# B&R Automation Studio project Vrtalka
Automation Studio 4.2.10.53 SP

## Configuration HW_config

### Task classes (Cpu.sw)
```
Cyclic#4 (cycle 100000 us, tolerance 100000 us):
  Vrtalka <- Vrtalka.prg
VcDataObjects: Vrtalk <- HMI.VrtalkaHMI.dob
```

### Hardware
```
4PPC70_101G_20B : 4PPC70.101G-20B v1.4.0.0
  Connector IF2:
    ActivateDevice = 1
    HostName = arsim
    Vnc1
    VncKeyMappingFile1 = VC\PS2-Keyboard1.dis
    VncMaxConnections1 = 2
    VncRefreshRate1 = 100
    VncTitle1 = HMIvrt
  ConfigurationID = Vrtalka_HW_config
  Simulation = 1
  Connections = 5
  TimerDeviceType = SWIOTIMER
  Cyclic1Duration = 10000
  Cyclic1Tolerance = 10000
  Cyclic2Duration = 20000
  Cyclic2Tolerance = 20000
  Cyclic3Duration = 50000
  Cyclic3Tolerance = 50000
  Cyclic4Duration = 100000
  Cyclic4Tolerance = 100000
  Cyclic5Duration = 200000
  Cyclic5Tolerance = 200000
  Cyclic6Duration = 500000
  Cyclic6Tolerance = 500000
  Cyclic7Duration = 1000000
  Cyclic7Tolerance = 1000000
  Cyclic8Duration = 10000
  Cyclic8Tolerance = 30000000
  VcObjectName = Vrtalk
  KeyMappingFile = VC\4PPC70_101G_20B.dis
```

## Configuration SimConf

CPU 4PPC70.101G-20B, AutomationRuntime D4.26, Build 4.1.2, Vc V4.26.5

### Task classes (Cpu.sw)
```
Cyclic#4:
  programHMI <- HMI.programHMI.prg [disabled]
Cyclic#7:
  Vrtalka <- Vrtalka.prg [disabled]
VcDataObjects: Vrtalk <- HMI.VrtalkaHMI.dob
Binaries: vcfile, vcrt, vctcal, vcfntttf, vcctext, arial, vcalarm, vcmgr, vccovl, vccnum, vcpfar00, vcdsint, vcpdvnc, vccslider, vcshared, vcpdsw, seguisb, vccbtn, Vrtalk03, vccstr, vcgclass, vcdsloc, arialbd, vcnet, TCData, segoeuib, segoeui, vccbmp, vcbclass, vccline, solid4n6, Vrtalk02, Vrtalk01, vccshape, User, ashwd, arconfig, sysconf, Role, asfw, iomap, Vrtal103, Vrtal102, vcpkat
Libraries: fileio, asieccon, dataobj, vcresman, astime, runtime
```

## Configuration SimulationConfig

CPU 4PPC70.101G-20B, AutomationRuntime D4.26, Build 4.1.2, Vc V4.26.5

### Task classes (Cpu.sw)
```
Cyclic#4 (cycle 100000 us, tolerance 100000 us):
  Program <- Program.prg
VcDataObjects: Vrtalk <- VrtalkaHMI.dob
Binaries: vcmgr, vcpfar00, arialbd, vcpdsw, vcalarm, vcshared, vcnet, vcgclass, vctcal, Vrtalk01, TCData, vcpdvnc, vccnum, Vrtalk02, vcfntttf, vcctext, Vrtalk03, vcdsint, vcfile, vcpkat, vcrt, vcbclass, vcdsloc, vccovl, arial, vccslider, vccbtn, reemkz6g, vccbmp, vccline, ashwd, User, sysconf, asfw, arconfig, iomap, Role, vccbar
Libraries: MTBasics, brsystem, MTTypes, sys_lib, runtime, fileio, vcresman, dataobj, asieccon, astime
```

### Hardware
```
4PPC70_101G_20B : 4PPC70.101G-20B v1.4.0.0
  Connector IF2:
    ActivateDevice = 1
    HostName = vrtalkahmi
    Vnc1
    VncVcObjectName1 = Vrtalk
    VncKeyMappingFile1 = VC\PS2-Keyboard.dis
    VncRefreshRate1 = 100
    VncTitle1 = Vrtalka
  ConfigurationID = Vrtalka_Config1
  TimerDeviceType = SWIOTIMER
  Cyclic1Duration = 10000
  Cyclic1Tolerance = 10000
  Cyclic2Duration = 20000
  Cyclic2Tolerance = 20000
  Cyclic3Duration = 50000
  Cyclic3Tolerance = 50000
  Cyclic4Duration = 100000
  Cyclic4Tolerance = 100000
  Cyclic5Duration = 200000
  Cyclic5Tolerance = 200000
  Cyclic6Duration = 500000
  Cyclic6Tolerance = 500000
  Cyclic7Duration = 1000000
  Cyclic7Tolerance = 1000000
  Cyclic8Duration = 10000
  Cyclic8Tolerance = 30000000
  KeyMappingFile = VC\4PPC70_101G_20B.dis
```

## Logical view

Binary libraries used (declarations not repeated): operator, runtime, astime, AsIecCon, MTBasics 2.30.0, brsystem, MTTypes 1.03.4, sys_lib


### Program Logical/Vrtalka (IEC)

#### AGR_Actions.st
```iecst
ACTION SomeTestAction:
	diHMIin2 := TRUE;
END_ACTION

ACTION SetInitialAgrValues:
	// Nastavi sirine agregatov
	agr1.agr_width := 30;
	agr2.agr_width := 30;
	agr3.agr_width := 30;
	agr4.agr_width := 30;
	agr5.agr_width := 30;
	agr6.agr_width := 30;

	// Nastavi minimalne pozicje agregatov
	agr1.poz_agr_min := agr1.agr_width;
	agr2.poz_agr_min := agr1.poz_agr_min + agr2.agr_width;
	agr3.poz_agr_min := agr2.poz_agr_min + agr3.agr_width;
	agr4.poz_agr_min := agr3.poz_agr_min + agr4.agr_width;
	agr5.poz_agr_min := agr4.poz_agr_min + agr5.agr_width;
	agr6.poz_agr_min := agr5.poz_agr_min + agr6.agr_width;

	// Reset nastavljenih pozicj
	agr1.poz_agr_s := 0;
	agr2.poz_agr_s := 0;
	agr3.poz_agr_s := 0;
	agr4.poz_agr_s := 0;
	agr5.poz_agr_s := 0;
	agr6.poz_agr_s := 0;

	// Reset trenutnih pozicij
	agr1.poz_agr_a := 0;
	agr2.poz_agr_a := 0;
	agr3.poz_agr_a := 0;
	agr4.poz_agr_a := 0;
	agr5.poz_agr_a := 0;
	agr6.poz_agr_a := 0;

	// Reset okej boolov
	agr1.agr_pos_ok := FALSE;
	agr2.agr_pos_ok := FALSE;
	agr3.agr_pos_ok := FALSE;
	agr4.agr_pos_ok := FALSE;
	agr5.agr_pos_ok := FALSE;
	agr6.agr_pos_ok := FALSE;

	// Reset ali je agr aktiven
	agr1.agr_active := FALSE;
	agr2.agr_active := FALSE;
	agr3.agr_active := FALSE;
	agr4.agr_active := FALSE;
	agr5.agr_active := FALSE;
	agr6.agr_active := FALSE;

	// Nastavi status agregata
	agr1.ag_status := 0;
	agr2.ag_status := 0;
	agr3.ag_status := 0;
	agr4.ag_status := 0;
	agr5.ag_status := 0;
	agr6.ag_status := 0;

END_ACTION

ACTION SetMaxAgrValues:  (* Izracun trenutnih maksimalnih pozicij *)

END_ACTION

// Sprosti zavore na agregatih
ACTION ReleaseAgrBrakes:
	ZavoraAgregata(agr1, FALSE);
	ZavoraAgregata(agr2, FALSE);
	ZavoraAgregata(agr3, FALSE);
	ZavoraAgregata(agr4, FALSE);
	ZavoraAgregata(agr5, FALSE);
	ZavoraAgregata(agr6, FALSE);

END_ACTION

ACTION LockAgrBrakes:
	ZavoraAgregata(agr1, TRUE);
	ZavoraAgregata(agr2, TRUE);
	ZavoraAgregata(agr3, TRUE);
	ZavoraAgregata(agr4, TRUE);
	ZavoraAgregata(agr5, TRUE);
	ZavoraAgregata(agr6, TRUE);

END_ACTION

ACTION SetHomePosAgr: (* Vse agregate peljemo na minimalne pozicije *)
	(*
	Nastaviti se morajo naslednje spremenljivke
	agr<#>.poz_agr_s - vozicke prepeljemo v minimalne lege dolocene v spremenljivki agr<#>.poz_agr_min
	agr<#>.poz_agr_a - dejanske pozicije agregatov (agregati so skupaj in naslonjeni, izracuna se iz sirine agregatov)
	agr<#>.poz_agr_i - izhodiscna pozicija agregata, ce zelimo kasneje popraviti lego, peljemo v HOME in nazaj razporedimo
	*)
	// Pomaknemo vozicek v max ce se ni
	PomikVozicka(1000, vozicek);
	// Iztegnemo zaklep na vozicku
	ZaklepAgregata(vozicek, TRUE);
	// Pomaknemo vozicek iz maksimuma v minimalno lego agregata 6 - agregati se med seboj dotikajo)
	PomikVozicka(agr6.poz_agr_min, vozicek);

	// Nastavimo status vozicka
	agr1.ag_status := 3;
	agr2.ag_status := 3;
	agr3.ag_status := 3;
	agr4.ag_status := 3;
	agr5.ag_status := 3;
	agr6.ag_status := 3;

	// Pozicije agregatov so sedaj znane
	// Agr1
	agr1.ag_status := 2;
	agr1.poz_agr_s := agr1.poz_agr_min;
	agr1.poz_agr_a := agr1.poz_agr_s;
	agr1.poz_agr_i := agr1.poz_agr_a;
	agr1.agr_pos_ok := TRUE;
	// Agr 2
	agr2.ag_status := 2;
	agr2.poz_agr_s := agr2.poz_agr_min;
	agr2.poz_agr_a := agr2.poz_agr_s;
	agr2.poz_agr_i := agr2.poz_agr_a;
	agr2.agr_pos_ok := TRUE;
	// Agr 3
	agr3.ag_status := 2;
	agr3.poz_agr_s := agr3.poz_agr_min;
	agr3.poz_agr_a := agr3.poz_agr_s;
	agr3.poz_agr_i := agr3.poz_agr_a;
	agr3.agr_pos_ok := TRUE;
	// Agr 4
	agr4.ag_status := 2;
	agr4.poz_agr_s := agr4.poz_agr_min;
	agr4.poz_agr_a := agr4.poz_agr_s;
	agr4.poz_agr_i := agr4.poz_agr_a;
	agr4.agr_pos_ok := TRUE;
	// Agr 5
	agr5.ag_status := 2;
	agr5.poz_agr_s := agr5.poz_agr_min;
	agr5.poz_agr_a := agr5.poz_agr_s;
	agr5.poz_agr_i := agr5.poz_agr_a;
	agr5.agr_pos_ok := TRUE;
	// Agr 6
	agr6.ag_status := 2;
	agr6.poz_agr_s := agr6.poz_agr_min;
	agr6.poz_agr_a := agr6.poz_agr_s;
	agr6.poz_agr_i := agr6.poz_agr_a;
	agr6.agr_pos_ok := TRUE;

END_ACTION

ACTION SetIzbraniAgrVal: (* Nastavljanje spremenljivke izbrani_agr iz boolov aktivnih agr *)

	// Za vsak agregat se preveri ce je aktiviran in ce je ustrezen bit v spremenljivki izbrani_agr postavljen na 1
	IF (agr1.agr_active = TRUE) AND (izbrani_agr.0 = 0) THEN
		izbrani_agr.0 := 1;
	ELSIF (agr1.agr_active = FALSE) AND (izbrani_agr.0 = 1) THEN
		izbrani_agr.0 := 0;
	END_IF;

	IF (agr2.agr_active = TRUE) AND (izbrani_agr.1 = 0) THEN
		izbrani_agr.1 := 1;
	ELSIF (agr2.agr_active = FALSE) AND (izbrani_agr.1 = 1) THEN
		izbrani_agr.1 := 0;
	END_IF;

	IF (agr3.agr_active = TRUE) AND (izbrani_agr.2 = 0) THEN
		izbrani_agr.2 := 1;
	ELSIF (agr3.agr_active = FALSE) AND (izbrani_agr.2 = 1) THEN
		izbrani_agr.2 := 0;
	END_IF;

	IF (agr4.agr_active = TRUE) AND (izbrani_agr.3 = 0) THEN
		izbrani_agr.3 := 1;
	ELSIF (agr4.agr_active = FALSE) AND (izbrani_agr.3 = 1) THEN
		izbrani_agr.3 := 0;
	END_IF;

	IF (agr5.agr_active = TRUE) AND (izbrani_agr.4 = 0) THEN
		izbrani_agr.4 := 1;
	ELSIF (agr5.agr_active = FALSE) AND (izbrani_agr.4 = 1) THEN
		izbrani_agr.4 := 0;
	END_IF;

	IF (agr6.agr_active = TRUE) AND (izbrani_agr.5 = 0) THEN
		izbrani_agr.5 := 1;
	ELSIF (agr6.agr_active = FALSE) AND (izbrani_agr.5 = 1) THEN
		izbrani_agr.5 := 0;
	END_IF;

END_ACTION
```

#### SRV_Actions.st
```iecst
ACTION SetInitialSrvValues:
	// Relevatne vrednosti pozicij
	vozicek.poz_srv_max := 1000;
	vozicek.poz_srv_min := agr1.poz_agr_min;

	// Reset ostalih spremenljivk

	// Zaklep agregata noter (Varnost)
	ZaklepAgregata(vozicek, FALSE);
	TestZaklepaAgr(vozicek);

	vozicek.servo_act := 0;
	vozicek.servo_set := 0;

	vozicek.servo_in_pos := FALSE;
	vozicek.servo_moving := FALSE;

	// Zaklep agregata noter ter pomik v skrajno lego
	PomikVozicka(n_pos := vozicek.poz_srv_max, vozicek := vozicek);
END_ACTION
```

#### General_actions.st
```iecst
ACTION ReadVarsFromHMI: (* Preberi vse spremenljivke iz HMI ekrana *)
	// Dummy
	diHMIin1 := diHMIin1;

	// Agregat
	agr1.agr_active := agr1.agr_active;
	agr2.agr_active := agr2.agr_active;
	agr3.agr_active := agr3.agr_active;
	agr4.agr_active := agr4.agr_active;
	agr5.agr_active := agr5.agr_active;
	agr6.agr_active := agr6.agr_active;

	SetIzbraniAgrVal;

	agr1.poz_agr_s := agr1.poz_agr_s;
	agr2.poz_agr_s := agr2.poz_agr_s;
	agr3.poz_agr_s := agr3.poz_agr_s;
	agr4.poz_agr_s := agr4.poz_agr_s;
	agr5.poz_agr_s := agr5.poz_agr_s;
	agr6.poz_agr_s := agr6.poz_agr_s;

END_ACTION
```

#### PROC_actions.st
```iecst
ACTION makeStep:
	WHILE diSTEP = FALSE DO
	END_WHILE;
	diSTEP := FALSE;
END_ACTION

ACTION nastavljanjeAgregatov:

	// Preveri ce so vse pozicije agregatov znane
	diPozAgrOK := agr1.agr_pos_ok AND agr2.agr_pos_ok AND agr3.agr_pos_ok AND agr4.agr_pos_ok AND agr5.agr_pos_ok AND agr6.agr_pos_ok;
	SetIzbraniAgrVal;
	makeStep;
	IF diPozAgrOK = FALSE THEN
		SetHomePosAgr;
	END_IF;
	makeStep;
	IF currentPage <> 20 THEN
		changePage := 20;
	END_IF;

	makeStep;

	// Pocakaj za vsak slucaj da se odpre nastavitven ekran
	WHILE currentPage <> 20 DO
	END_WHILE;
	sistemskoObvestilo := 'Stroj v nastavljanju';

	WHILE diShraniPozicije = FALSE DO
	END_WHILE;
	ReadVarsFromHMI;
	popupConfirm := 0;

	WHILE diPotrdiPozicije = FALSE DO
	END_WHILE;

	diShraniPozicije := FALSE;
	diPotrdiPozicije := FALSE;
	popupConfirm := 1;

	// Stroj je pripravljen na delo, nastavitve agregatov so potrjene
	// Stroj je priprvljen na uporabo
	doStrojPripravljen := TRUE;

	WHILE diStartStroja = FALSE DO
	END_WHILE;

	//popupWarning := 1;
	changePage := 10;

END_ACTION

ACTION OperacijaVrtanja: (* mock operacija za vrtanje *)
	// Tukaj bi prisla koda za dejansko vrtanje vrtalke
END_ACTION
```

#### Cyclic.st - Cyclic code
```iecst
PROGRAM _CYCLIC
	// Preveri ali je stroj pripravljen na delovanje
	IF doStrojPripravljen = FALSE THEN
		nastavljanjeAgregatov;
	ELSIF (diStartStroja = TRUE OR doDelovanje = TRUE) AND doStrojPripravljen = TRUE THEN
		sistemskoObvestilo := 'Stroj v delovanju';
		doDelovanje := TRUE;
		diStartStroja := FALSE;
		OperacijaVrtanja;
	ELSIF diPrekiniCikel = TRUE AND doDelovanje = TRUE THEN
		sistemskoObvestilo := 'Stroj v zaustavljanju';
		OperacijaVrtanja;
		doDelovanje := FALSE;
		sistemskoObvestilo := 'Stroj zaustavljen';
	END_IF;

END_PROGRAM
```

#### Init.st - Init code
```iecst
PROGRAM _INIT

	//Nastavi trenutno stran na Settings ob zagonu
	changePage := 0;
	sistemskoObvestilo := 'ZAGON STROJA';
	// Resetiraj pozicije in spremenljivke agregatov
	SetInitialAgrValues;
	ReleaseAgrBrakes;
	WHILE diGoHome = FALSE DO
	END_WHILE;

	// Zapri okno
	popupWarning := 1;
	// Resetiraj spremenljivke vozicka in ga zapelji v max lego
	SetInitialSrvValues;
	// Postavi agregate v HOME pozicijo
	SetHomePosAgr;
	diGoHome := FALSE;
END_PROGRAM
```

#### HMIVars.var
```iecst
VAR
	setupScreen : BOOL := FALSE; (*Ali je setup screen aktiven*)
END_VAR
```

### VrtalkaVars.var - Local variables
```iecst
(*Delovne variable*)
VAR
	sistemskoObvestilo : STRING[80] := 'Ni obvestil'; (*spremenljivka za obvestila*)
END_VAR
(*HMI variable*)
VAR
	changePage : UINT := 0; (*spremenljivka za prikaz popupa*)
	popupConfirm : UINT := 0; (*Spremenljivka za pop-up okno ob potrditvi*)
	popupWarning : UINT := 0; (*Spremenljivka za pop-up okno ob zagonu*)
END_VAR
VAR CONSTANT
	settingsPage : UINT := 20; (*Index nastavitvene strani*)
END_VAR
VAR
	currentPage : UINT := 0; (*Spremenljivka ali je setupScreen aktiven*)
END_VAR
(*Agregati*)
VAR
	agr1 : agr_typ := (izbrani_agr_mask:=1); (*agregat 1*)
	agr2 : agr_typ := (izbrani_agr_mask:=2); (*agregat 2*)
	agr3 : agr_typ := (izbrani_agr_mask:=4); (*agregat 3*)
	agr4 : agr_typ := (izbrani_agr_mask:=8); (*agregat 4*)
	agr5 : agr_typ := (izbrani_agr_mask:=16); (*agregat 5*)
	agr6 : agr_typ := (izbrani_agr_mask:=32); (*agregat 6*)
	diPozAgrOK : BOOL; (*ali so pozicije agregatov znane*)
	diHMIin1 : BOOL := FALSE;
	diHMIin2 : BOOL := FALSE;
END_VAR
(*GhostVars [DI/DO]*)
VAR
	diSTEP : BOOL := FALSE; (*Spremenljivka za step-anje*)
	diPrekiniCikel : BOOL := FALSE; (*Prekinitev cikla*)
	diSoftStop : BOOL := FALSE; (*ustavitev delovanja*)
	diStartStroja : BOOL := FALSE; (*digital input za start Stroja*)
	doDelovanje : BOOL := FALSE; (*stroj je v delovanju*)
	diRand : BOOL := FALSE; (*DI random*)
	diSetAgrPoz : BOOL := FALSE; (*DI za pomik agregatov v nastavljene pozicije*)
	diGoHome : BOOL := FALSE; (*DI za homing vozickov -> poz_agr_min*)
	doFunSuccess : BOOL := FALSE; (*Mock HMI prikaz *)
	doHMIout1 : BOOL := FALSE;
	diPotrdiPozicije : BOOL := FALSE; (*shrani in potrdi pozicije*)
	diShraniPozicije : BOOL := FALSE; (*potrdi pozicije agregatov*)
	doStrojPripravljen : BOOL := FALSE; (*stroj je pripravljen za delo*)
	izbrani_agr : UINT := 0; (*int izbranih agregatov*)
END_VAR
(*Nastavljene pozicije agregatov [REAL/D]*)
VAR
	poz_agr_i : REAL := 0.0; (*Skupna sirina agregatov -> izracuna iz st. agregatov in njihove sirine*)
END_VAR
(*Agregati varnostne spemenljivke [REAL]*)
VAR CONSTANT
	raz_agr : REAL := 30; (*Minimalen razmik agregatov, izhaja iz sirine agregatov*)
END_VAR
(*Servo*)
VAR
	vozicek : servo_typ := (0); (*Spremenljivka za servo typ*)
END_VAR
```

### Types.typ
```iecst
TYPE
	agr_typ : 	STRUCT
		poz_agr_s : REAL := 0; (*Nastavljena pozicija agregata*)
		poz_agr_a : REAL := 0; (*Dejanska pozicija agregata*)
		poz_agr_i : REAL; (*Izhodiscna pozicija agregata*)
		poz_agr_min : REAL := 0; (*Minimalna skrajna lega agregata*)
		poz_agr_max : REAL := 0; (*Maksimalna skrajna lega agregata*)
		agr_pos_ok : BOOL := FALSE; (*Agregat v poziciji*)
		o_agr_zav : BOOL := FALSE; (*Zavora agregata*)
		agr_width : REAL := 30; (*Sirina agregata*)
		agr_active : BOOL := FALSE; (*Ali je agregat aktiven*)
		izbrani_agr_mask : UINT; (*Maska za spremenljivko izbrani agregat*)
		ag_status : UINT;
	END_STRUCT;
	servo_typ : 	STRUCT
		servo_set : REAL := 0; (*Nastavljena pozicija servo motorja*)
		servo_act : REAL := 0; (*Trenutna pozicija servo motorja*)
		servo_in_pos : BOOL := FALSE; (*Servo na poziciji*)
		o_agr_zak_z : BOOL := FALSE; (*Razmik agr. -> zaklep ZUNAJ ; OUTPUT*)
		o_agr_zak_o : BOOL := FALSE; (*Razmik agr. -> zaklep NOTER ; OUTPUT*)
		i_agr_zak_z : BOOL := FALSE; (*Razmik agr. -> zaklep ZUNAJ ; INPUT*)
		i_agr_zak_o : BOOL := FALSE; (*Razmik agr. -> zaklep NOTER ; INPUT*)
		poz_srv_max : REAL := 1000; (*Maksimalna pozicija servota*)
		poz_srv_min : REAL := 0; (*Minimalna pozicija servota*)
		servo_moving : BOOL := FALSE; (*DO da se servo premika*)
		agr_zak : BOOL := FALSE; (*ali je agregat zaklnjen (TRUE je, FALSE ni)*)
	END_STRUCT;
END_TYPE
```

- Visualisation Logical/HMI/VrtalkaHMI (not shown)

### Program Logical/HMI/programHMI (IEC)

#### Main.st - Init, cyclic, exit code
```iecst
PROGRAM _INIT
	(* Insert code here *)
	//obvestiloHMI := 'INIT UFNKCIJA';
	popupWarning := 0;
	WHILE diGoHome = FALSE DO
	END_WHILE;
	changePage := 20;
	// Zapri okno
	popupWarning := 1;
END_PROGRAM

PROGRAM _CYCLIC
	(* Insert code here *)
	//obvestiloHMI := 'CIKLIK';
	(* Insert code here *)
	//poz_agr1_a := poz_agr1_a + 5;
	stevec := stevec + 1;
	//changePage := 10;
	ReadVarsFromHMI;

END_PROGRAM

PROGRAM _EXIT
	(* Insert code here *)
	obvestiloHMI := 'ENDER';

END_PROGRAM
```

#### Variables.var - Local variables
```iecst
VAR
	obvestiloHMI : STRING[80] := 'prazno';
	stevec : UINT := 0;
END_VAR
```

#### HMI_actions.st
```iecst
ACTION ReadVarsFromHMI: (* Preberi vse spremenljivke iz HMI ekrana *)
	// Dummy
	diHMIin1 := diHMIin1;

	// Agregat
	agr1 := agr1;
	agr2 := agr2;
	agr3 := agr3;
	agr4 := agr4;
	agr5 := agr5;
	agr6 := agr6;

	diPozAgrOK := diPozAgrOK;

	diSTEP := diSTEP;
	diPrekiniCikel := diPrekiniCikel;
	diSoftStop := diSoftStop;
	diStartStroja := diStartStroja;
	doDelovanje := doDelovanje;
	diRand := diRand;
	diSetAgrPoz := diSetAgrPoz;
	diGoHome := diGoHome;
	doFunSuccess := doFunSuccess;
	doHMIout1 := doHMIout1;
	diPotrdiPozicije := diPotrdiPozicije;
	diShraniPozicije := diShraniPozicije;
	doStrojPripravljen := doStrojPripravljen;
	izbrani_agr := izbrani_agr;

	vozicek := vozicek;

	diHMIin1 := diHMIin1;
	diHMIin2 := diHMIin2;

	(*
	agr1.agr_active := agr1.agr_active;
	agr2.agr_active := agr2.agr_active;
	agr3.agr_active := agr3.agr_active;
	agr4.agr_active := agr4.agr_active;
	agr5.agr_active := agr5.agr_active;
	agr6.agr_active := agr6.agr_active;

	agr1.poz_agr_s := agr1.poz_agr_s;
	agr2.poz_agr_s := agr2.poz_agr_s;
	agr3.poz_agr_s := agr3.poz_agr_s;
	agr4.poz_agr_s := agr4.poz_agr_s;
	agr5.poz_agr_s := agr5.poz_agr_s;
	agr6.poz_agr_s := agr6.poz_agr_s;
	*)
END_ACTION
```

### hmiVariables.var - not listed in the package file held
```iecst
VAR
	hmiPageVar : USINT := 10;
END_VAR
```

### Program Logical/Program (IEC)

#### Variables.var - Local variables
```iecst
(*Delovne variable*)
(*Agregati*)
VAR
	agr1 : agr_typ := (izbrani_agr_mask:=1); (*agregat 1*)
	agr2 : agr_typ := (izbrani_agr_mask:=2); (*agregat 2*)
	agr3 : agr_typ := (izbrani_agr_mask:=4); (*agregat 3*)
	agr4 : agr_typ := (izbrani_agr_mask:=8); (*agregat 4*)
	agr5 : agr_typ := (izbrani_agr_mask:=16); (*agregat 5*)
	agr6 : agr_typ := (izbrani_agr_mask:=32); (*agregat 6*)
	diHMIin1 : BOOL := FALSE;
	diHMIin2 : BOOL := FALSE;
END_VAR
(*GhostVars [DI/DO]*)
VAR
	diPrekiniCikel : BOOL := FALSE; (*Prekinitev cikla*)
	diSoftStop : BOOL := FALSE; (*ustavitev delovanja*)
	diStartStroja : BOOL := FALSE; (*digital input za start Stroja*)
	doDelovanje : BOOL := FALSE; (*stroj je v delovanju*)
	diRand : BOOL := FALSE; (*DI random*)
	diSetAgrPoz : BOOL := FALSE; (*DI za pomik agregatov v nastavljene pozicije*)
	diGoHome : BOOL := FALSE; (*DI za homing vozickov -> poz_agr_min*)
	doFunSuccess : BOOL := FALSE; (*Mock HMI prikaz *)
	doHMIout1 : BOOL := FALSE;
	doStrojPripravljen : BOOL := FALSE; (*stroj je pripravljen za delo*)
	izbrani_agr : UINT := 0; (*int izbranih agregatov*)
END_VAR
(*Nastavljene pozicije agregatov [REAL/D]*)
VAR
	poz_agr_i : REAL := 0.0; (*Skupna sirina agregatov -> izracuna iz st. agregatov in njihove sirine*)
END_VAR
(*Agregati varnostne spemenljivke [REAL]*)
VAR CONSTANT
	raz_agr : REAL := 30; (*Minimalen razmik agregatov, izhaja iz sirine agregatov*)
END_VAR
(*Servo*)
VAR
	vozicek : servo_typ := (0); (*Spremenljivka za servo typ*)
END_VAR
```

#### Types.typ
```iecst
TYPE
	agr_typ : 	STRUCT
		poz_agr_s : REAL := 0; (*Nastavljena pozicija agregata*)
		poz_agr_a : REAL := 0; (*Dejanska pozicija agregata*)
		poz_agr_min : REAL := 0; (*Minimalna skrajna lega agregata*)
		poz_agr_max : REAL := 0; (*Maksimalna skrajna lega agregata*)
		agr_pos_ok : BOOL := FALSE; (*Agregat v poziciji*)
		o_agr_zav : BOOL := FALSE; (*Zavora agregata*)
		agr_width : REAL := 30; (*Sirina agregata*)
		agr_active : BOOL := FALSE; (*Ali je agregat aktiven*)
		izbrani_agr_mask : UINT; (*Maska za spremenljivko izbrani agregat*)
	END_STRUCT;
	servo_typ : 	STRUCT
		servo_set : REAL := 0; (*Nastavljena pozicija servo motorja*)
		servo_act : REAL := 0; (*Trenutna pozicija servo motorja*)
		servo_in_pos : BOOL := FALSE; (*Servo na poziciji*)
		o_agr_zak_z : BOOL := FALSE; (*Razmik agr. -> zaklep ZUNAJ ; OUTPUT*)
		o_agr_zak_o : BOOL := FALSE; (*Razmik agr. -> zaklep NOTER ; OUTPUT*)
		i_agr_zak_z : BOOL := FALSE; (*Razmik agr. -> zaklep ZUNAJ ; INPUT*)
		i_agr_zak_o : BOOL := FALSE; (*Razmik agr. -> zaklep NOTER ; INPUT*)
		poz_srv_max : REAL := 1000; (*Maksimalna pozicija servota*)
		poz_srv_min : REAL := 0; (*Minimalna pozicija servota*)
		servo_moving : BOOL := FALSE; (*DO da se servo premika*)
		agr_zak : BOOL := FALSE; (*ali je agregat zaklnjen (TRUE je, FALSE ni)*)
	END_STRUCT;
END_TYPE
```

#### AGR_Actions.st
```iecst
ACTION SomeTestAction:
	diHMIin2 := TRUE;
END_ACTION

ACTION SetInitialAgrValues:
	// Nastavi sirine agregatov
	agr1.agr_width := 30;
	agr2.agr_width := 30;
	agr3.agr_width := 30;
	agr4.agr_width := 30;
	agr5.agr_width := 30;
	agr6.agr_width := 30;

	// Nastavi minimalne pozicje agregatov
	agr1.poz_agr_min := agr1.agr_width;
	agr2.poz_agr_min := agr1.poz_agr_min + agr2.agr_width;
	agr3.poz_agr_min := agr2.poz_agr_min + agr3.agr_width;
	agr4.poz_agr_min := agr3.poz_agr_min + agr4.agr_width;
	agr5.poz_agr_min := agr4.poz_agr_min + agr5.agr_width;
	agr6.poz_agr_min := agr5.poz_agr_min + agr6.agr_width;

	// Reset nastavljenih pozicj
	agr1.poz_agr_s := 0;
	agr2.poz_agr_s := 0;
	agr3.poz_agr_s := 0;
	agr4.poz_agr_s := 0;
	agr5.poz_agr_s := 0;
	agr6.poz_agr_s := 0;

	// Reset trenutnih pozicij
	agr1.poz_agr_a := 0;
	agr2.poz_agr_a := 0;
	agr3.poz_agr_a := 0;
	agr4.poz_agr_a := 0;
	agr5.poz_agr_a := 0;
	agr6.poz_agr_a := 0;

	// Reset okej boolov
	agr1.agr_pos_ok := FALSE;
	agr2.agr_pos_ok := FALSE;
	agr3.agr_pos_ok := FALSE;
	agr4.agr_pos_ok := FALSE;
	agr5.agr_pos_ok := FALSE;
	agr6.agr_pos_ok := FALSE;

	// Reset ali je agr aktiven
	agr1.agr_active := FALSE;
	agr2.agr_active := FALSE;
	agr3.agr_active := FALSE;
	agr4.agr_active := FALSE;
	agr5.agr_active := FALSE;
	agr6.agr_active := FALSE;

END_ACTION

ACTION SetMaxAgrValues:  (* Izracun trenutnih maksimalnih pozicij *)

END_ACTION

// Sprosti zavore na agregatih
ACTION ReleaseAgrBrakes:
	ZavoraAgregata(agr1, FALSE);
	ZavoraAgregata(agr2, FALSE);
	ZavoraAgregata(agr3, FALSE);
	ZavoraAgregata(agr4, FALSE);
	ZavoraAgregata(agr5, FALSE);
	ZavoraAgregata(agr6, FALSE);

END_ACTION

ACTION SetHomePosAgr: (* Vse agregate peljemo na minimalne pozicije *)
	// Pomaknemo vozicek v max ce se ni
	PomikVozicka(1000, vozicek);
	// Iztegnemo zaklep na vozicku
	ZaklepAgregata(vozicek, TRUE);
	// Pomaknemo vozicek iz maksimuma v minimalno lego agregata 6 - agregati se med seboj dotikajo)
	PomikVozicka(agr6.poz_agr_min, vozicek);

	// Pozicije agregatov so sedaj znane
	// Agr1
	agr1.poz_agr_s := agr1.poz_agr_min;
	agr1.poz_agr_a := agr1.poz_agr_min;
	agr1.agr_pos_ok := TRUE;
	// Agr 2
	agr2.poz_agr_s := agr2.poz_agr_min;
	agr2.poz_agr_a := agr2.poz_agr_min;
	agr2.agr_pos_ok := TRUE;
	// Agr 3
	agr3.poz_agr_s := agr3.poz_agr_min;
	agr3.poz_agr_a := agr3.poz_agr_min;
	agr3.agr_pos_ok := TRUE;
	// Agr 4
	agr4.poz_agr_s := agr4.poz_agr_min;
	agr4.poz_agr_a := agr4.poz_agr_min;
	agr4.agr_pos_ok := TRUE;
	// Agr 5
	agr5.poz_agr_s := agr5.poz_agr_min;
	agr5.poz_agr_a := agr5.poz_agr_min;
	agr5.agr_pos_ok := TRUE;
	// Agr 6
	agr6.poz_agr_s := agr6.poz_agr_min;
	agr6.poz_agr_a := agr6.poz_agr_min;
	agr6.agr_pos_ok := TRUE;

END_ACTION

ACTION SetIzbraniAgrVal: (* Nastavljanje spremenljivke izbrani_agr iz boolov aktivnih agr *)

	//izbrani_agr := 666;
	IF (agr1.agr_active = TRUE) AND ((izbrani_agr AND 2#0000_0000_0000_0001) = FALSE) THEN
		izbrani_agr := izbrani_agr OR 2#0000_0000_0000_0001;
	END_IF
	IF (agr1.agr_active = FALSE) AND ((izbrani_agr AND 2#0000_0000_0000_0001) = TRUE) THEN
		izbrani_agr := izbrani_agr XOR 2#0000_0000_0000_0001;
	END_IF

	IF (agr2.agr_active = TRUE) AND ((izbrani_agr AND 2#0000_0000_0000_0010) = FALSE) THEN
		izbrani_agr := izbrani_agr OR 2#0000_0000_0000_0010;
	END_IF
	IF (agr2.agr_active = FALSE) AND ((izbrani_agr AND 2#0000_0000_0000_0010) = TRUE) THEN
		izbrani_agr := izbrani_agr XOR 2#0000_0000_0000_0010;
	END_IF
		(*
	IF agr1.agr_active = TRUE THEN
		izbrani_agr := izbrani_agr OR 2#0000_0000_0000_0001;
	END_IF;
	IF agr1.agr_active = FALSE THEN
		izbrani_agr := izbrani_agr XOR 2#0000_0000_0000_0001;
	END_IF;

	IF agr2.agr_active = TRUE THEN
		izbrani_agr := izbrani_agr OR 2#0000_0000_0000_0010;
	END_IF;
	IF agr1.agr_active = FALSE THEN
		izbrani_agr := izbrani_agr XOR 2#0000_0000_0000_0010;
	END_IF;

	IF agr3.agr_active = TRUE THEN
		izbrani_agr := izbrani_agr OR 2#0000_0000_0000_0100;
	ELSE
		izbrani_agr := izbrani_agr XOR 2#0000_0000_0000_0100;
	END_IF;

	IF agr4.agr_active = TRUE THEN
		izbrani_agr := izbrani_agr OR 2#0000_0000_0000_1000;
	ELSE
		izbrani_agr := izbrani_agr XOR 2#0000_0000_0000_1000;
	END_IF;

	IF agr5.agr_active = TRUE THEN
		izbrani_agr := izbrani_agr OR 2#0000_0000_0001_0000;
	ELSE
		izbrani_agr := izbrani_agr XOR 2#0000_0000_0001_0000;
	END_IF;

	IF agr6.agr_active = TRUE THEN
		izbrani_agr := izbrani_agr OR 2#0000_0000_0010_0000;
	ELSE
		izbrani_agr := izbrani_agr XOR 2#0000_0000_0010_0000;
	END_IF;
	*)
END_ACTION
```

#### General_actions.st
```iecst
ACTION ReadVarsFromHMI:
	diHMIin1 := diHMIin1;
	(*
	agr1.agr_active := agr1.agr_active;
	agr2.agr_active := agr2.agr_active;
	agr3.agr_active := agr3.agr_active;
	agr4.agr_active := agr4.agr_active;
	agr5.agr_active := agr5.agr_active;
	agr6.agr_active := agr6.agr_active;
	*)

END_ACTION
```

#### Cyclic.st
```iecst
PROGRAM _CYCLIC
	(* Insert code here *)
	//poz_agr1_a := poz_agr1_a + 5;
	ReadVarsFromHMI;
	vozicek.servo_set := vozicek.servo_set;
	IF diStartStroja THEN
		agr1.poz_agr_a := agr1.poz_agr_a + 5;

		PomikVozicka(n_pos := vozicek.servo_set, vozicek := vozicek);
		SomeTestAction;

		// Dodatek iz vscode
		doDelovanje := TRUE;
	ELSE
		doDelovanje := FALSE;
	END_IF;

	//izbrani_agr := izbrani_agr + 1;

	// Using variables from HMI to set actual vars

	IF diHMIin1 = TRUE THEN
		SetIzbraniAgrVal;
	END_IF;

	//ZaklepAgregata(vozicek := vozicek, zak_agr := diHMIin1);
	//TestZaklepaAgr(vozicek := vozicek);

END_PROGRAM
```

#### Exit.st
```iecst
PROGRAM _EXIT
	(* Insert code here *)

END_PROGRAM
```

#### Init.st
```iecst
PROGRAM _INIT

	// Resetiraj pozicije in spremenljivke agregatov
	SetInitialAgrValues;
	ReleaseAgrBrakes;

	// Resetiraj spremenljivke vozicka in ga zapelji v max lego
	SetInitialSrvValues;

	WHILE diGoHome = FALSE DO
	END_WHILE;

	// Postavi agregate v HOME pozicijo
	SetHomePosAgr;
	diGoHome := FALSE;

	// Stroj je priprvljen na uporabo
	doStrojPripravljen := TRUE;

END_PROGRAM
```

#### VrtalkaFunctions.st
```iecst
FUNCTION TestZaklepaAgr (* Funkcija za preverjanje zaklepa agregata *)
	IF vozicek.i_agr_zak_z = TRUE AND vozicek.i_agr_zak_o = FALSE THEN
		vozicek.agr_zak := FALSE;
		TestZaklepaAgr := TRUE;
	ELSIF vozicek.i_agr_zak_z = FALSE AND vozicek.i_agr_zak_o = TRUE THEN
		vozicek.agr_zak := TRUE;
		TestZaklepaAgr := TRUE;
	ELSE
		//  Zaradi varnosti privzamemo da je zaklep zunaj
		vozicek.agr_zak := TRUE;
		TestZaklepaAgr := FALSE;
	END_IF
END_FUNCTION

FUNCTION ZaklepAgregata (* Funckija za zaklep agregata|| TRUE->zaklep ; FALSE-> odklep *)
	IF zak_agr = TRUE THEN
		vozicek.o_agr_zak_o := TRUE;
		vozicek.o_agr_zak_z := FALSE;
		vozicek.i_agr_zak_o := vozicek.o_agr_zak_o;
		vozicek.i_agr_zak_z := vozicek.o_agr_zak_z;
		ZaklepAgregata := vozicek.i_agr_zak_o AND NOT vozicek.i_agr_zak_z;
	ELSIF zak_agr = FALSE THEN

		vozicek.o_agr_zak_o := FALSE;
		vozicek.o_agr_zak_z := TRUE;
		vozicek.i_agr_zak_o := vozicek.o_agr_zak_o;
		vozicek.i_agr_zak_z := vozicek.o_agr_zak_z;
		vozicek.agr_zak := FALSE;
		ZaklepAgregata := NOT vozicek.i_agr_zak_o AND vozicek.i_agr_zak_z;
	ELSE
		ZaklepAgregata := FALSE;
	END_IF;
END_FUNCTION

FUNCTION PomikVozicka (* Funkcija za pomik vozicka, REAL je zeljena pozicija *)
	vozicek.servo_set := n_pos;

	IF  vozicek.servo_act > vozicek.servo_set THEN
		n_pomik := -1;
	ELSIF vozicek.servo_act < vozicek.servo_set THEN
		n_pomik := 1;
	ELSE
		//
		vozicek.servo_in_pos := TRUE;
		PomikVozicka := TRUE;
	END_IF;

	WHILE vozicek.servo_act <> vozicek.servo_set DO
		vozicek.servo_moving := TRUE;
		vozicek.servo_act := vozicek.servo_act + n_pomik;
	END_WHILE
	vozicek.servo_moving := FALSE;
	// preverjanje ali je vozicek na ustreznem mestu
	// ce je
	IF vozicek.servo_act = vozicek.servo_set THEN
		vozicek.servo_in_pos := TRUE;
		PomikVozicka := TRUE;
		// Ce ni na ustreznem mestu vrzemo vn false funkcije
	ELSE
		vozicek.servo_in_pos := FALSE;
		PomikVozicka := FALSE;
	END_IF
END_FUNCTION

FUNCTION ZavoraAgregata (* Funckija za zaklep in odklep agregata *)
	agr.o_agr_zav := agr_zav;
	ZavoraAgregata := TRUE;
END_FUNCTION
```

#### VrtalkaFunctions.fun
```iecst
FUNCTION ZaklepAgregata : BOOL (*TRUE -> success, FALSE -> failure*)
	VAR_INPUT
		vozicek : servo_typ;
		zak_agr : BOOL; (*TRUE -> iztegni zaklep, FALSE -> skrci zaklep*)
	END_VAR
END_FUNCTION

FUNCTION TestZaklepaAgr : BOOL (*Funkcija za preverjanje zaklepa agregata*)
	VAR_INPUT
		vozicek : servo_typ; (*input tipa*)
	END_VAR
END_FUNCTION

FUNCTION PomikVozicka : BOOL (*Funkcija za pomik vozicka*)
	VAR_INPUT
		n_pos : REAL; (*Nova pozicija servota*)
		vozicek : servo_typ; (*Passamo spremenljivko v funkcijo da lahko prirejamo vrednsti*)
	END_VAR
	VAR
		n_pomik : REAL; (*pomik v plus ali minus odvisno od servo_act >< == servo_set*)
	END_VAR
END_FUNCTION

FUNCTION ZavoraAgregata : BOOL (*Funkcija za sprostitev ali  zaklep zavore*)
	VAR_INPUT
		agr : agr_typ; (*Spremenljivka za agregat -> pass reference*)
		agr_zav : BOOL; (*TRUE -> Aktiviraj zavoro, FALSE -> sprosti zavoro*)
	END_VAR
END_FUNCTION
```

Listed in the project but not available here: Logical/Vrtalka/ST_src/Exit.st, Logical/Vrtalka/VrtalkaFunctions.st, Logical/Vrtalka/VrtalkaFunctions.fun, Logical/HMI/programHMI/Types.typ, Logical/Program/Vrtalka_actions/SRV_Actions.st
